# EPICS substitutions: IOCs/12id/iocBoot/ioc12ida2/canberra_13.substitutions
file "$(MCA)/mcaApp/Db/simple_mca.db"
{
pattern
{P           M       DTYP           INP         PREC  CHANS}
{12ida2:med:   mca1  "asynMCA"   "@asyn(AIM2/1 0)"    3  2048}
{12ida2:med:   mca2  "asynMCA"   "@asyn(AIM2/1 1)"    3  2048}
{12ida2:med:   mca3  "asynMCA"   "@asyn(AIM2/1 2)"    3  2048}
{12ida2:med:   mca4  "asynMCA"   "@asyn(AIM2/2 0)"    3  2048}
{12ida2:med:   mca5  "asynMCA"   "@asyn(AIM2/2 1)"    3  2048}
{12ida2:med:   mca6  "asynMCA"   "@asyn(AIM2/2 2)"    3  2048}
{12ida2:med:   mca7  "asynMCA"   "@asyn(AIM3/1 0)"    3  2048}
{12ida2:med:   mca8  "asynMCA"   "@asyn(AIM3/1 1)"    3  2048}
{12ida2:med:   mca9  "asynMCA"   "@asyn(AIM3/1 2)"    3  2048}
{12ida2:med:   mca10 "asynMCA"   "@asyn(AIM3/2 0)"    3  2048}
{12ida2:med:   mca11 "asynMCA"   "@asyn(AIM3/3 1)"    3  2048}
{12ida2:med:   mca12 "asynMCA"   "@asyn(AIM3/4 2)"    3  2048}
{12ida2:med:   mca13 "asynMCA"   "@asyn(AIM3/2 3)"    3  2048}
{12ida2:med:   mca0  "Soft Channel"   ""     3  2048}
}

file "$(MCA)/mcaApp/Db/icb_amp.db"
{
pattern
{P			AMP		PORT}
{12ida2:med:	amp1	"icbAmp1"}
{12ida2:med:	amp2	"icbAmp2"}
{12ida2:med:	amp3	"icbAmp3"}
{12ida2:med:	amp4	"icbAmp4"}
{12ida2:med:	amp5	"icbAmp5"}
{12ida2:med:	amp6	"icbAmp6"}
{12ida2:med:	amp7	"icbAmp7"}
{12ida2:med:	amp8	"icbAmp8"}
{12ida2:med:	amp9	"icbAmp9"}
{12ida2:med:	amp10	"icbAmp10"}
{12ida2:med:	amp11	"icbAmp11"}
{12ida2:med:	amp12	"icbAmp12"}
{12ida2:med:	amp13	"icbAmp13"}
}

file "$(MCA)/mcaApp/Db/icb_adc.db"
{
pattern
{P			ADC		PORT}
{12ida2:med:	adc1	"icbAdc1"}
{12ida2:med:	adc2	"icbAdc2"}
{12ida2:med:	adc3	"icbAdc3"}
{12ida2:med:	adc4	"icbAdc4"}
}

file "$(MCA)/mcaApp/Db/icb_hvps.db"
{
pattern
{P			HVPS	LIMIT	PORT}
{12ida2:med:	hvps1	1000	"icbHvps1"}
}
